TYPE ST_TestSuiteResults :
STRUCT
    // General test results
    NumberOfTestSuites : UINT; // The total number of test suites
    NumberOfTestCases : UDINT; // The total number of test cases (for all test suites)
    NumberOfSuccessfulTestCases : UDINT; // The total number of test cases that had all ASSERTS successful
    NumberOfFailedTestCases : UDINT; // The total number of test cases that had at least one ASSERT failed
    NumberOfSkippedTestCases : UDINT; // The total number of test cases that were skipped (disabled)
    Duration : LREAL; // Duration it took for all test suites to finish, in seconds

    // Test results for each individiual test suite
    TestSuiteResults : ARRAY[1..GVL_Param_TcUnit.MaxNumberOfTestSuites] OF ST_TestSuiteResult;
END_STRUCT
END_TYPE

(* stored: Version 1.1.0.1
   DUT ST_TestSuiteResults: Id {9853f266-188f-4741-a381-36145196003d} *)
